    |   movel([0.283198, -1.182378, -2.685957, -0.844054, 1.570796, 1.853994],accel_mss,speed_ms,0,blend_radius_m)
    |   movel([0.283190, -1.181681, -2.686275, -0.844433, 1.570796, 1.853986],accel_mss,speed_ms,0,blend_radius_m)
    |   movel([0.283388, -1.180979, -2.686595, -0.844815, 1.570796, 1.854185],accel_mss,speed_ms,0,blend_radius_m)
    |   movel([0.283803, -1.180261, -2.686921, -0.845207, 1.570796, 1.854599],accel_mss,speed_ms,0,blend_radius_m)
    |   movel([0.284097, -1.179507, -2.687264, -0.845619, 1.570796, 1.854893],accel_mss,speed_ms,0,blend_radius_m)
    |   movel([0.284020, -1.179269, -2.687371, -0.845748, 1.570796, 1.854816],accel_mss,speed_ms,0,blend_radius_m)
    |   movel([0.283537, -1.179119, -2.687439, -0.845830, 1.570796, 1.854333],accel_mss,speed_ms,0,blend_radius_m)
    |   movel([0.283308, -1.178461, -2.687737, -0.846191, 1.570796, 1.854105],accel_mss,speed_ms,0,blend_radius_m)
    |   movel([0.283133, -1.176565, -2.688593, -0.847230, 1.570796, 1.853929],accel_mss,speed_ms,0,blend_radius_m)
    |   movel([0.283249, -1.175411, -2.689113, -0.847866, 1.570796, 1.854045],accel_mss,speed_ms,0,blend_radius_m)
    |   movel([0.283954, -1.172938, -2.690220, -0.849231, 1.570796, 1.854751],accel_mss,speed_ms,0,blend_radius_m)
    |   movel([0.284534, -1.171660, -2.690790, -0.849939, 1.570796, 1.855330],accel_mss,speed_ms,0,blend_radius_m)
    |   movel([0.286108, -1.169102, -2.691926, -0.851361, 1.570796, 1.856905],accel_mss,speed_ms,0,blend_radius_m)
    |   movel([0.287085, -1.167859, -2.692475, -0.852054, 1.570796, 1.857881],accel_mss,speed_ms,0,blend_radius_m)
    |   movel([0.288923, -1.165863, -2.693354, -0.853171, 1.570796, 1.859719],accel_mss,speed_ms,0,blend_radius_m)
    |   movel([0.289212, -1.165437, -2.693541, -0.853410, 1.570796, 1.860008],accel_mss,speed_ms,0,blend_radius_m)
    |   movel([0.289229, -1.165158, -2.693664, -0.853567, 1.570796, 1.860026],accel_mss,speed_ms,0,blend_radius_m)
    |   movel([0.288991, -1.164941, -2.693759, -0.853689, 1.570796, 1.859788],accel_mss,speed_ms,0,blend_radius_m)
    |   movel([0.288746, -1.164927, -2.693765, -0.853697, 1.570796, 1.859543],accel_mss,speed_ms,0,blend_radius_m)
    |   movel([0.288455, -1.165081, -2.693698, -0.853610, 1.570796, 1.859252],accel_mss,speed_ms,0,blend_radius_m)
    |   movel([0.287437, -1.165989, -2.693299, -0.853101, 1.570796, 1.858234],accel_mss,speed_ms,0,blend_radius_m)
    |   movel([0.286224, -1.167338, -2.692705, -0.852345, 1.570796, 1.857020],accel_mss,speed_ms,0,blend_radius_m)
    |   movel([0.285012, -1.168950, -2.691993, -0.851446, 1.570796, 1.855809],accel_mss,speed_ms,0,blend_radius_m)
    |   movel([0.283819, -1.170819, -2.691165, -0.850406, 1.570796, 1.854615],accel_mss,speed_ms,0,blend_radius_m)
    |   movel([0.282921, -1.172578, -2.690381, -0.849430, 1.570796, 1.853718],accel_mss,speed_ms,0,blend_radius_m)
    |   movel([0.282300, -1.174282, -2.689619, -0.848488, 1.570796, 1.853096],accel_mss,speed_ms,0,blend_radius_m)
    |   movel([0.281922, -1.175986, -2.688854, -0.847549, 1.570796, 1.852719],accel_mss,speed_ms,0,blend_radius_m)
    |   movel([0.281810, -1.177316, -2.688255, -0.846818, 1.570796, 1.852606],accel_mss,speed_ms,0,blend_radius_m)
    |   movel([0.281869, -1.178652, -2.687651, -0.846086, 1.570796, 1.852665],accel_mss,speed_ms,0,blend_radius_m)
    |   movel([0.282044, -1.179763, -2.687147, -0.845479, 1.570796, 1.852840],accel_mss,speed_ms,0,blend_radius_m)
    |   movel([0.282451, -1.180138, -2.686977, -0.845274, 1.570796, 1.853247],accel_mss,speed_ms,0,blend_radius_m)
    |   movel([0.282464, -1.180320, -2.686894, -0.845174, 1.570796, 1.853260],accel_mss,speed_ms,0,blend_radius_m)
    |   movel([0.281904, -1.182146, -2.686063, -0.844180, 1.570796, 1.852701],accel_mss,speed_ms,0,blend_radius_m)
    |   movel([0.281872, -1.183086, -2.685633, -0.843670, 1.570796, 1.852669],accel_mss,speed_ms,0,blend_radius_m)
    |   movel([0.282108, -1.183902, -2.685260, -0.843227, 1.570796, 1.852905],accel_mss,speed_ms,0,blend_radius_m)
    |   movel([0.282593, -1.184554, -2.684961, -0.842874, 1.570796, 1.853389],accel_mss,speed_ms,0,blend_radius_m)
    |   movel([0.283618, -1.185190, -2.684669, -0.842530, 1.570796, 1.854415],accel_mss,speed_ms,0,blend_radius_m)
    |   movel([0.284266, -1.185300, -2.684618, -0.842471, 1.570796, 1.855062],accel_mss,speed_ms,0,blend_radius_m)
    |   movel([0.285735, -1.185305, -2.684616, -0.842468, 1.570796, 1.856532],accel_mss,speed_ms,0,blend_radius_m)
    |   movel([0.286093, -1.185248, -2.684642, -0.842499, 1.570796, 1.856889],accel_mss,speed_ms,0,blend_radius_m)
    |   movel([0.286619, -1.184980, -2.684765, -0.842644, 1.570796, 1.857415],accel_mss,speed_ms,0,blend_radius_m)
    |   movel([0.286888, -1.184698, -2.684895, -0.842796, 1.570796, 1.857685],accel_mss,speed_ms,0,blend_radius_m)
    |   movel([0.287131, -1.184139, -2.685151, -0.843099, 1.570796, 1.857927],accel_mss,speed_ms,0,blend_radius_m)
    |   movel([0.287047, -1.183997, -2.685216, -0.843176, 1.570796, 1.857843],accel_mss,speed_ms,0,blend_radius_m)
    |   movel([0.285248, -1.183986, -2.685221, -0.843182, 1.570796, 1.856044],accel_mss,speed_ms,0,blend_radius_m)
    |   speed_ms = 0.005
    |   movel([0.285248, -1.174261, -2.680335, -0.857793, 1.570796, 1.856044],accel_mss,speed_ms,0,blend_radius_m)
    |   speed_ms = 0.040
    |   movel([0.315314, -1.140804, -2.694900, -0.876685, 1.570796, 1.886110],accel_mss,speed_ms,0,blend_radius_m)
    |   speed_ms = 0.005
    |   movel([0.315314, -1.150611, -2.699936, -0.861843, 1.570796, 1.886110],accel_mss,speed_ms,0,blend_radius_m)
    |   speed_ms = 0.025
    |   movel([0.314615, -1.150672, -2.699910, -0.861807, 1.570796, 1.885411],accel_mss,speed_ms,0,blend_radius_m)
    |   movel([0.314030, -1.150638, -2.699924, -0.861827, 1.570796, 1.884826],accel_mss,speed_ms,0,blend_radius_m)
    |   movel([0.311693, -1.150473, -2.699994, -0.861922, 1.570796, 1.882489],accel_mss,speed_ms,0,blend_radius_m)
    |   movel([0.309738, -1.150673, -2.699909, -0.861807, 1.570796, 1.880534],accel_mss,speed_ms,0,blend_radius_m)
    |   movel([0.307713, -1.151133, -2.699714, -0.861542, 1.570796, 1.878509],accel_mss,speed_ms,0,blend_radius_m)
    |   movel([0.305786, -1.151819, -2.699423, -0.861147, 1.570796, 1.876582],accel_mss,speed_ms,0,blend_radius_m)
    |   movel([0.303092, -1.153186, -2.698841, -0.860362, 1.570796, 1.873888],accel_mss,speed_ms,0,blend_radius_m)
    |   movel([0.300320, -1.155004, -2.698064, -0.859321, 1.570796, 1.871116],accel_mss,speed_ms,0,blend_radius_m)
    |   movel([0.297716, -1.157102, -2.697163, -0.858123, 1.570796, 1.868512],accel_mss,speed_ms,0,blend_radius_m)
    |   movel([0.295514, -1.159300, -2.696215, -0.856874, 1.570796, 1.866310],accel_mss,speed_ms,0,blend_radius_m)
    |   movel([0.294232, -1.160879, -2.695531, -0.855979, 1.570796, 1.865028],accel_mss,speed_ms,0,blend_radius_m)
    |   movel([0.293549, -1.162093, -2.695003, -0.855293, 1.570796, 1.864346],accel_mss,speed_ms,0,blend_radius_m)
    |   movel([0.293356, -1.163124, -2.694554, -0.854711, 1.570796, 1.864153],accel_mss,speed_ms,0,blend_radius_m)
    |   movel([0.293601, -1.164123, -2.694117, -0.854149, 1.570796, 1.864397],accel_mss,speed_ms,0,blend_radius_m)
    |   movel([0.293780, -1.164753, -2.693841, -0.853795, 1.570796, 1.864576],accel_mss,speed_ms,0,blend_radius_m)
    |   movel([0.293763, -1.165466, -2.693529, -0.853394, 1.570796, 1.864560],accel_mss,speed_ms,0,blend_radius_m)
    |   movel([0.293570, -1.166121, -2.693241, -0.853027, 1.570796, 1.864367],accel_mss,speed_ms,0,blend_radius_m)
    |   movel([0.293220, -1.166587, -2.693036, -0.852766, 1.570796, 1.864016],accel_mss,speed_ms,0,blend_radius_m)
    |   movel([0.292642, -1.167187, -2.692772, -0.852430, 1.570796, 1.863438],accel_mss,speed_ms,0,blend_radius_m)
    |   movel([0.292135, -1.167909, -2.692454, -0.852027, 1.570796, 1.862932],accel_mss,speed_ms,0,blend_radius_m)
    |   movel([0.291374, -1.169709, -2.691657, -0.851023, 1.570796, 1.862170],accel_mss,speed_ms,0,blend_radius_m)
    |   movel([0.291099, -1.170961, -2.691101, -0.850327, 1.570796, 1.861895],accel_mss,speed_ms,0,blend_radius_m)
    |   movel([0.291056, -1.172041, -2.690621, -0.849728, 1.570796, 1.861852],accel_mss,speed_ms,0,blend_radius_m)
    |   movel([0.291248, -1.172980, -2.690201, -0.849207, 1.570796, 1.862045],accel_mss,speed_ms,0,blend_radius_m)
    |   movel([0.292278, -1.174667, -2.689447, -0.848276, 1.570796, 1.863075],accel_mss,speed_ms,0,blend_radius_m)
    |   movel([0.291718, -1.176581, -2.688586, -0.847222, 1.570796, 1.862514],accel_mss,speed_ms,0,blend_radius_m)
    |   movel([0.291364, -1.178095, -2.687903, -0.846391, 1.570796, 1.862160],accel_mss,speed_ms,0,blend_radius_m)
    |   movel([0.291302, -1.179246, -2.687382, -0.845761, 1.570796, 1.862098],accel_mss,speed_ms,0,blend_radius_m)
    |   movel([0.291534, -1.180211, -2.686944, -0.845234, 1.570796, 1.862330],accel_mss,speed_ms,0,blend_radius_m)
    |   movel([0.292084, -1.181146, -2.686519, -0.844725, 1.570796, 1.862881],accel_mss,speed_ms,0,blend_radius_m)
    |   movel([0.292452, -1.181723, -2.686256, -0.844410, 1.570796, 1.863248],accel_mss,speed_ms,0,blend_radius_m)
    |   movel([0.292557, -1.182195, -2.686040, -0.844154, 1.570796, 1.863353],accel_mss,speed_ms,0,blend_radius_m)
    |   movel([0.292420, -1.182572, -2.685868, -0.843948, 1.570796, 1.863216],accel_mss,speed_ms,0,blend_radius_m)
    |   movel([0.292084, -1.182881, -2.685727, -0.843781, 1.570796, 1.862880],accel_mss,speed_ms,0,blend_radius_m)
    |   movel([0.291599, -1.182907, -2.685715, -0.843767, 1.570796, 1.862395],accel_mss,speed_ms,0,blend_radius_m)
    |   movel([0.290967, -1.182262, -2.686010, -0.844117, 1.570796, 1.861763],accel_mss,speed_ms,0,blend_radius_m)
    |   movel([0.290399, -1.181349, -2.686426, -0.844614, 1.570796, 1.861195],accel_mss,speed_ms,0,blend_radius_m)
    |   movel([0.290052, -1.180315, -2.686897, -0.845177, 1.570796, 1.860849],accel_mss,speed_ms,0,blend_radius_m)
    |   movel([0.289921, -1.178962, -2.687510, -0.845916, 1.570796, 1.860717],accel_mss,speed_ms,0,blend_radius_m)
    |   movel([0.290018, -1.178289, -2.687815, -0.846285, 1.570796, 1.860815],accel_mss,speed_ms,0,blend_radius_m)
    |   movel([0.290598, -1.175773, -2.688950, -0.847666, 1.570796, 1.861395],accel_mss,speed_ms,0,blend_radius_m)
    |   movel([0.290557, -1.175356, -2.689137, -0.847896, 1.570796, 1.861354],accel_mss,speed_ms,0,blend_radius_m)
    |   movel([0.289995, -1.174027, -2.689733, -0.848629, 1.570796, 1.860791],accel_mss,speed_ms,0,blend_radius_m)
    |   movel([0.289750, -1.173019, -2.690184, -0.849186, 1.570796, 1.860546],accel_mss,speed_ms,0,blend_radius_m)
    |   movel([0.289679, -1.171982, -2.690647, -0.849760, 1.570796, 1.860475],accel_mss,speed_ms,0,blend_radius_m)
    |   movel([0.289783, -1.170857, -2.691148, -0.850385, 1.570796, 1.860579],accel_mss,speed_ms,0,blend_radius_m)
    |   movel([0.290038, -1.169795, -2.691619, -0.850975, 1.570796, 1.860835],accel_mss,speed_ms,0,blend_radius_m)
    |   movel([0.290466, -1.168697, -2.692105, -0.851587, 1.570796, 1.861262],accel_mss,speed_ms,0,blend_radius_m)
    |   movel([0.291014, -1.167717, -2.692538, -0.852134, 1.570796, 1.861811],accel_mss,speed_ms,0,blend_radius_m)
    |   movel([0.291733, -1.166783, -2.692950, -0.852656, 1.570796, 1.862529],accel_mss,speed_ms,0,blend_radius_m)
    |   movel([0.292496, -1.165923, -2.693328, -0.853138, 1.570796, 1.863292],accel_mss,speed_ms,0,blend_radius_m)
    |   movel([0.292182, -1.164857, -2.693796, -0.853736, 1.570796, 1.862978],accel_mss,speed_ms,0,blend_radius_m)
    |   movel([0.292034, -1.163840, -2.694241, -0.854308, 1.570796, 1.862830],accel_mss,speed_ms,0,blend_radius_m)
    |   movel([0.292166, -1.162774, -2.694706, -0.854908, 1.570796, 1.862963],accel_mss,speed_ms,0,blend_radius_m)
    |   movel([0.292594, -1.161641, -2.695200, -0.855548, 1.570796, 1.863391],accel_mss,speed_ms,0,blend_radius_m)
    |   movel([0.293313, -1.160418, -2.695731, -0.856240, 1.570796, 1.864110],accel_mss,speed_ms,0,blend_radius_m)
    |   movel([0.294423, -1.159056, -2.696321, -0.857012, 1.570796, 1.865219],accel_mss,speed_ms,0,blend_radius_m)
    |   movel([0.296451, -1.157016, -2.697201, -0.858172, 1.570796, 1.867248],accel_mss,speed_ms,0,blend_radius_m)
    |   movel([0.298621, -1.155009, -2.698062, -0.859318, 1.570796, 1.869417],accel_mss,speed_ms,0,blend_radius_m)
    |   movel([0.300305, -1.153670, -2.698634, -0.860084, 1.570796, 1.871101],accel_mss,speed_ms,0,blend_radius_m)
    |   movel([0.302226, -1.152415, -2.699170, -0.860805, 1.570796, 1.873022],accel_mss,speed_ms,0,blend_radius_m)
    |   movel([0.304176, -1.151356, -2.699619, -0.861413, 1.570796, 1.874972],accel_mss,speed_ms,0,blend_radius_m)
    |   movel([0.306205, -1.150461, -2.699999, -0.861929, 1.570796, 1.877001],accel_mss,speed_ms,0,blend_radius_m)
    |   movel([0.308208, -1.149771, -2.700291, -0.862327, 1.570796, 1.879004],accel_mss,speed_ms,0,blend_radius_m)
    |   movel([0.310151, -1.149301, -2.700490, -0.862598, 1.570796, 1.880947],accel_mss,speed_ms,0,blend_radius_m)
    |   movel([0.312023, -1.149055, -2.700594, -0.862740, 1.570796, 1.882819],accel_mss,speed_ms,0,blend_radius_m)
    |   movel([0.313699, -1.149054, -2.700594, -0.862741, 1.570796, 1.884495],accel_mss,speed_ms,0,blend_radius_m)
    |   movel([0.315241, -1.149302, -2.700489, -0.862597, 1.570796, 1.886037],accel_mss,speed_ms,0,blend_radius_m)
    |   movel([0.315653, -1.149518, -2.700398, -0.862473, 1.570796, 1.886449],accel_mss,speed_ms,0,blend_radius_m)
    |   movel([0.315810, -1.149883, -2.700244, -0.862262, 1.570796, 1.886606],accel_mss,speed_ms,0,blend_radius_m)
    |   movel([0.315675, -1.150279, -2.700076, -0.862034, 1.570796, 1.886471],accel_mss,speed_ms,0,blend_radius_m)
    |   movel([0.315314, -1.150611, -2.699936, -0.861843, 1.570796, 1.886110],accel_mss,speed_ms,0,blend_radius_m)
    |   movel([0.314615, -1.150672, -2.699910, -0.861807, 1.570796, 1.885411],accel_mss,speed_ms,0,blend_radius_m)
    |   movel([0.314030, -1.150638, -2.699924, -0.861827, 1.570796, 1.884826],accel_mss,speed_ms,0,blend_radius_m)
    |   movel([0.312501, -1.150532, -2.699969, -0.861888, 1.570796, 1.883297],accel_mss,speed_ms,0,blend_radius_m)
    |   speed_ms = 0.005
    |   movel([0.312501, -1.140725, -2.694933, -0.876731, 1.570796, 1.883297],accel_mss,speed_ms,0,blend_radius_m)
    |   speed_ms = 0.040
    |   movel([0.330564, -1.150947, -2.690604, -0.870838, 1.570796, 1.901361],accel_mss,speed_ms,0,blend_radius_m)
    |   speed_ms = 0.005
    |   movel([0.330564, -1.160732, -2.695595, -0.856062, 1.570796, 1.901361],accel_mss,speed_ms,0,blend_radius_m)
    |   speed_ms = 0.025
    |   movel([0.330341, -1.160709, -2.695605, -0.856075, 1.570796, 1.901138],accel_mss,speed_ms,0,blend_radius_m)
    |   movel([0.329903, -1.160225, -2.695815, -0.856349, 1.570796, 1.900699],accel_mss,speed_ms,0,blend_radius_m)
    |   movel([0.327422, -1.156688, -2.697342, -0.858359, 1.570796, 1.898218],accel_mss,speed_ms,0,blend_radius_m)
    |   movel([0.325962, -1.154973, -2.698077, -0.859338, 1.570796, 1.896758],accel_mss,speed_ms,0,blend_radius_m)
    |   movel([0.324619, -1.153780, -2.698588, -0.860022, 1.570796, 1.895416],accel_mss,speed_ms,0,blend_radius_m)
    |   movel([0.323055, -1.152831, -2.698992, -0.860565, 1.570796, 1.893851],accel_mss,speed_ms,0,blend_radius_m)
    |   movel([0.321507, -1.152257, -2.699237, -0.860895, 1.570796, 1.892303],accel_mss,speed_ms,0,blend_radius_m)
    |   movel([0.319774, -1.151965, -2.699361, -0.861063, 1.570796, 1.890571],accel_mss,speed_ms,0,blend_radius_m)
    |   movel([0.317908, -1.151964, -2.699361, -0.861064, 1.570796, 1.888704],accel_mss,speed_ms,0,blend_radius_m)
    |   movel([0.315914, -1.152256, -2.699237, -0.860896, 1.570796, 1.886710],accel_mss,speed_ms,0,blend_radius_m)
    |   movel([0.313852, -1.152813, -2.699000, -0.860576, 1.570796, 1.884648],accel_mss,speed_ms,0,blend_radius_m)
    |   movel([0.312994, -1.153164, -2.698850, -0.860374, 1.570796, 1.883791],accel_mss,speed_ms,0,blend_radius_m)
    |   movel([0.309997, -1.154816, -2.698145, -0.859428, 1.570796, 1.880794],accel_mss,speed_ms,0,blend_radius_m)
    |   movel([0.308659, -1.155885, -2.697687, -0.858818, 1.570796, 1.879456],accel_mss,speed_ms,0,blend_radius_m)
    |   movel([0.307739, -1.157048, -2.697187, -0.858154, 1.570796, 1.878535],accel_mss,speed_ms,0,blend_radius_m)
    |   movel([0.307072, -1.158460, -2.696578, -0.857351, 1.570796, 1.877868],accel_mss,speed_ms,0,blend_radius_m)
    |   movel([0.306749, -1.159391, -2.696176, -0.856822, 1.570796, 1.877546],accel_mss,speed_ms,0,blend_radius_m)
    |   movel([0.305275, -1.159870, -2.695969, -0.856551, 1.570796, 1.876072],accel_mss,speed_ms,0,blend_radius_m)
    |   movel([0.303894, -1.160437, -2.695723, -0.856229, 1.570796, 1.874691],accel_mss,speed_ms,0,blend_radius_m)
    |   movel([0.302617, -1.161210, -2.695387, -0.855792, 1.570796, 1.873414],accel_mss,speed_ms,0,blend_radius_m)
    |   movel([0.301445, -1.162187, -2.694962, -0.855240, 1.570796, 1.872242],accel_mss,speed_ms,0,blend_radius_m)
    |   movel([0.300377, -1.163363, -2.694449, -0.854576, 1.570796, 1.871173],accel_mss,speed_ms,0,blend_radius_m)
    |   movel([0.299472, -1.164674, -2.693876, -0.853839, 1.570796, 1.870268],accel_mss,speed_ms,0,blend_radius_m)
    |   movel([0.299212, -1.165270, -2.693615, -0.853504, 1.570796, 1.870008],accel_mss,speed_ms,0,blend_radius_m)
    |   movel([0.298716, -1.167186, -2.692772, -0.852431, 1.570796, 1.869512],accel_mss,speed_ms,0,blend_radius_m)
    |   movel([0.298670, -1.168206, -2.692322, -0.851861, 1.570796, 1.869466],accel_mss,speed_ms,0,blend_radius_m)
    |   movel([0.298783, -1.169018, -2.691963, -0.851408, 1.570796, 1.869580],accel_mss,speed_ms,0,blend_radius_m)
    |   movel([0.299074, -1.169391, -2.691798, -0.851200, 1.570796, 1.869871],accel_mss,speed_ms,0,blend_radius_m)
    |   movel([0.299181, -1.169609, -2.691701, -0.851078, 1.570796, 1.869978],accel_mss,speed_ms,0,blend_radius_m)
    |   movel([0.299059, -1.169979, -2.691538, -0.850873, 1.570796, 1.869855],accel_mss,speed_ms,0,blend_radius_m)
    |   movel([0.298029, -1.171218, -2.690987, -0.850184, 1.570796, 1.868826],accel_mss,speed_ms,0,blend_radius_m)
    |   movel([0.297342, -1.171992, -2.690642, -0.849755, 1.570796, 1.868138],accel_mss,speed_ms,0,blend_radius_m)
    |   movel([0.296221, -1.173730, -2.689866, -0.848793, 1.570796, 1.867017],accel_mss,speed_ms,0,blend_radius_m)
    |   movel([0.295912, -1.174497, -2.689523, -0.848369, 1.570796, 1.866708],accel_mss,speed_ms,0,blend_radius_m)
    |   movel([0.295851, -1.176623, -2.688567, -0.847199, 1.570796, 1.866647],accel_mss,speed_ms,0,blend_radius_m)
    |   movel([0.295881, -1.177717, -2.688074, -0.846598, 1.570796, 1.866678],accel_mss,speed_ms,0,blend_radius_m)
    |   movel([0.295853, -1.180600, -2.686767, -0.845022, 1.570796, 1.866650],accel_mss,speed_ms,0,blend_radius_m)
    |   movel([0.295776, -1.180820, -2.686667, -0.844902, 1.570796, 1.866573],accel_mss,speed_ms,0,blend_radius_m)
    |   movel([0.295324, -1.181183, -2.686502, -0.844704, 1.570796, 1.866120],accel_mss,speed_ms,0,blend_radius_m)
    |   movel([0.295147, -1.181242, -2.686475, -0.844672, 1.570796, 1.865943],accel_mss,speed_ms,0,blend_radius_m)
    |   movel([0.294864, -1.181150, -2.686517, -0.844722, 1.570796, 1.865660],accel_mss,speed_ms,0,blend_radius_m)
    |   movel([0.294694, -1.180670, -2.686735, -0.844984, 1.570796, 1.865490],accel_mss,speed_ms,0,blend_radius_m)
    |   movel([0.294468, -1.177649, -2.688104, -0.846635, 1.570796, 1.865265],accel_mss,speed_ms,0,blend_radius_m)
    |   movel([0.294543, -1.175723, -2.688972, -0.847694, 1.570796, 1.865339],accel_mss,speed_ms,0,blend_radius_m)
    |   movel([0.294956, -1.173994, -2.689748, -0.848647, 1.570796, 1.865752],accel_mss,speed_ms,0,blend_radius_m)
    |   movel([0.295721, -1.172423, -2.690450, -0.849516, 1.570796, 1.866517],accel_mss,speed_ms,0,blend_radius_m)
    |   movel([0.296837, -1.170971, -2.691097, -0.850321, 1.570796, 1.867633],accel_mss,speed_ms,0,blend_radius_m)
    |   movel([0.297554, -1.170204, -2.691438, -0.850748, 1.570796, 1.868351],accel_mss,speed_ms,0,blend_radius_m)
    |   movel([0.297337, -1.167906, -2.692455, -0.852028, 1.570796, 1.868133],accel_mss,speed_ms,0,blend_radius_m)
    |   movel([0.297604, -1.166489, -2.693079, -0.852821, 1.570796, 1.868400],accel_mss,speed_ms,0,blend_radius_m)
    |   movel([0.298106, -1.165037, -2.693717, -0.853635, 1.570796, 1.868903],accel_mss,speed_ms,0,blend_radius_m)
    |   movel([0.298782, -1.163781, -2.694267, -0.854341, 1.570796, 1.869579],accel_mss,speed_ms,0,blend_radius_m)
    |   movel([0.300034, -1.162202, -2.694956, -0.855231, 1.570796, 1.870830],accel_mss,speed_ms,0,blend_radius_m)
    |   movel([0.301657, -1.160695, -2.695611, -0.856083, 1.570796, 1.872454],accel_mss,speed_ms,0,blend_radius_m)
    |   movel([0.303428, -1.159450, -2.696151, -0.856789, 1.570796, 1.874224],accel_mss,speed_ms,0,blend_radius_m)
    |   movel([0.305117, -1.158647, -2.696498, -0.857245, 1.570796, 1.875913],accel_mss,speed_ms,0,blend_radius_m)
    |   movel([0.305966, -1.158277, -2.696657, -0.857454, 1.570796, 1.876763],accel_mss,speed_ms,0,blend_radius_m)
    |   movel([0.306111, -1.158107, -2.696731, -0.857551, 1.570796, 1.876908],accel_mss,speed_ms,0,blend_radius_m)
    |   movel([0.306523, -1.156986, -2.697214, -0.858190, 1.570796, 1.877319],accel_mss,speed_ms,0,blend_radius_m)
    |   movel([0.306747, -1.156613, -2.697374, -0.858402, 1.570796, 1.877544],accel_mss,speed_ms,0,blend_radius_m)
    |   movel([0.307476, -1.155654, -2.697785, -0.858949, 1.570796, 1.878273],accel_mss,speed_ms,0,blend_radius_m)
    |   movel([0.308347, -1.154796, -2.698153, -0.859440, 1.570796, 1.879144],accel_mss,speed_ms,0,blend_radius_m)
    |   movel([0.309487, -1.153902, -2.698535, -0.859951, 1.570796, 1.880283],accel_mss,speed_ms,0,blend_radius_m)
    |   movel([0.310666, -1.153129, -2.698865, -0.860395, 1.570796, 1.881462],accel_mss,speed_ms,0,blend_radius_m)
    |   movel([0.312068, -1.152374, -2.699187, -0.860828, 1.570796, 1.882864],accel_mss,speed_ms,0,blend_radius_m)
    |   movel([0.313470, -1.151766, -2.699446, -0.861178, 1.570796, 1.884266],accel_mss,speed_ms,0,blend_radius_m)
    |   movel([0.316489, -1.150865, -2.699828, -0.861696, 1.570796, 1.887286],accel_mss,speed_ms,0,blend_radius_m)
    |   movel([0.318328, -1.150563, -2.699956, -0.861870, 1.570796, 1.889125],accel_mss,speed_ms,0,blend_radius_m)
    |   movel([0.319922, -1.150503, -2.699981, -0.861905, 1.570796, 1.890719],accel_mss,speed_ms,0,blend_radius_m)
    |   movel([0.321440, -1.150681, -2.699906, -0.861802, 1.570796, 1.892236],accel_mss,speed_ms,0,blend_radius_m)
    |   movel([0.323038, -1.151114, -2.699722, -0.861553, 1.570796, 1.893835],accel_mss,speed_ms,0,blend_radius_m)
    |   movel([0.324964, -1.151992, -2.699349, -0.861048, 1.570796, 1.895760],accel_mss,speed_ms,0,blend_radius_m)
    |   movel([0.326646, -1.153232, -2.698822, -0.860336, 1.570796, 1.897442],accel_mss,speed_ms,0,blend_radius_m)
    |   movel([0.328267, -1.155000, -2.698066, -0.859323, 1.570796, 1.899063],accel_mss,speed_ms,0,blend_radius_m)
    |   movel([0.330866, -1.158912, -2.696383, -0.857094, 1.570796, 1.901662],accel_mss,speed_ms,0,blend_radius_m)
    |   movel([0.331156, -1.159778, -2.696008, -0.856603, 1.570796, 1.901953],accel_mss,speed_ms,0,blend_radius_m)
    |   movel([0.331017, -1.160335, -2.695767, -0.856287, 1.570796, 1.901813],accel_mss,speed_ms,0,blend_radius_m)
    |   movel([0.330564, -1.160732, -2.695595, -0.856062, 1.570796, 1.901361],accel_mss,speed_ms,0,blend_radius_m)
    |   movel([0.330341, -1.160709, -2.695605, -0.856075, 1.570796, 1.901138],accel_mss,speed_ms,0,blend_radius_m)
    |   movel([0.329903, -1.160225, -2.695815, -0.856349, 1.570796, 1.900699],accel_mss,speed_ms,0,blend_radius_m)
    |   movel([0.329043, -1.158994, -2.696348, -0.857047, 1.570796, 1.899840],accel_mss,speed_ms,0,blend_radius_m)
    |   speed_ms = 0.005
    |   movel([0.329043, -1.149205, -2.691349, -0.871835, 1.570796, 1.899840],accel_mss,speed_ms,0,blend_radius_m)
    |   speed_ms = 0.040
    |   movel([0.331713, -1.158475, -2.687349, -0.866565, 1.570796, 1.902510],accel_mss,speed_ms,0,blend_radius_m)
    |   speed_ms = 0.005
    |   movel([0.331713, -1.168242, -2.692306, -0.851841, 1.570796, 1.902510],accel_mss,speed_ms,0,blend_radius_m)
    |   speed_ms = 0.025
    |   movel([0.331306, -1.168113, -2.692363, -0.851912, 1.570796, 1.902103],accel_mss,speed_ms,0,blend_radius_m)
    |   movel([0.331181, -1.167790, -2.692506, -0.852093, 1.570796, 1.901977],accel_mss,speed_ms,0,blend_radius_m)
    |   movel([0.330488, -1.165082, -2.693697, -0.853610, 1.570796, 1.901285],accel_mss,speed_ms,0,blend_radius_m)
    |   movel([0.329418, -1.163092, -2.694568, -0.854729, 1.570796, 1.900215],accel_mss,speed_ms,0,blend_radius_m)
    |   movel([0.327976, -1.161415, -2.695298, -0.855676, 1.570796, 1.898772],accel_mss,speed_ms,0,blend_radius_m)
    |   movel([0.326286, -1.160232, -2.695812, -0.856345, 1.570796, 1.897083],accel_mss,speed_ms,0,blend_radius_m)
    |   movel([0.325017, -1.159721, -2.696033, -0.856635, 1.570796, 1.895813],accel_mss,speed_ms,0,blend_radius_m)
    |   movel([0.323332, -1.159309, -2.696211, -0.856869, 1.570796, 1.894129],accel_mss,speed_ms,0,blend_radius_m)
    |   movel([0.321666, -1.159053, -2.696322, -0.857014, 1.570796, 1.892462],accel_mss,speed_ms,0,blend_radius_m)
    |   movel([0.320604, -1.159119, -2.696294, -0.856976, 1.570796, 1.891400],accel_mss,speed_ms,0,blend_radius_m)
    |   movel([0.319128, -1.159715, -2.696036, -0.856638, 1.570796, 1.889924],accel_mss,speed_ms,0,blend_radius_m)
    |   movel([0.318351, -1.160251, -2.695804, -0.856335, 1.570796, 1.889148],accel_mss,speed_ms,0,blend_radius_m)
    |   movel([0.316474, -1.161927, -2.695075, -0.855386, 1.570796, 1.887270],accel_mss,speed_ms,0,blend_radius_m)
    |   movel([0.313923, -1.162515, -2.694819, -0.855054, 1.570796, 1.884719],accel_mss,speed_ms,0,blend_radius_m)
    |   movel([0.311493, -1.163182, -2.694529, -0.854679, 1.570796, 1.882289],accel_mss,speed_ms,0,blend_radius_m)
    |   movel([0.310725, -1.163546, -2.694369, -0.854473, 1.570796, 1.881521],accel_mss,speed_ms,0,blend_radius_m)
    |   movel([0.308314, -1.165097, -2.693690, -0.853601, 1.570796, 1.879110],accel_mss,speed_ms,0,blend_radius_m)
    |   movel([0.307457, -1.165878, -2.693348, -0.853163, 1.570796, 1.878254],accel_mss,speed_ms,0,blend_radius_m)
    |   movel([0.306883, -1.166716, -2.692979, -0.852694, 1.570796, 1.877680],accel_mss,speed_ms,0,blend_radius_m)
    |   movel([0.306453, -1.167771, -2.692514, -0.852104, 1.570796, 1.877249],accel_mss,speed_ms,0,blend_radius_m)
    |   movel([0.306245, -1.168703, -2.692103, -0.851583, 1.570796, 1.877041],accel_mss,speed_ms,0,blend_radius_m)
    |   movel([0.306317, -1.168871, -2.692028, -0.851490, 1.570796, 1.877113],accel_mss,speed_ms,0,blend_radius_m)
    |   movel([0.306750, -1.169089, -2.691932, -0.851368, 1.570796, 1.877546],accel_mss,speed_ms,0,blend_radius_m)
    |   movel([0.306794, -1.169237, -2.691866, -0.851286, 1.570796, 1.877590],accel_mss,speed_ms,0,blend_radius_m)
    |   movel([0.306593, -1.169712, -2.691656, -0.851021, 1.570796, 1.877390],accel_mss,speed_ms,0,blend_radius_m)
    |   movel([0.306273, -1.169988, -2.691533, -0.850867, 1.570796, 1.877070],accel_mss,speed_ms,0,blend_radius_m)
    |   movel([0.304136, -1.171018, -2.691076, -0.850295, 1.570796, 1.874933],accel_mss,speed_ms,0,blend_radius_m)
    |   movel([0.303280, -1.171628, -2.690804, -0.849956, 1.570796, 1.874076],accel_mss,speed_ms,0,blend_radius_m)
    |   movel([0.301531, -1.173235, -2.690087, -0.849066, 1.570796, 1.872327],accel_mss,speed_ms,0,blend_radius_m)
    |   movel([0.301020, -1.173828, -2.689822, -0.848738, 1.570796, 1.871816],accel_mss,speed_ms,0,blend_radius_m)
    |   movel([0.300389, -1.174911, -2.689337, -0.848141, 1.570796, 1.871186],accel_mss,speed_ms,0,blend_radius_m)
    |   movel([0.300062, -1.175767, -2.688952, -0.847669, 1.570796, 1.870858],accel_mss,speed_ms,0,blend_radius_m)
    |   movel([0.299607, -1.177615, -2.688120, -0.846654, 1.570796, 1.870404],accel_mss,speed_ms,0,blend_radius_m)
    |   movel([0.299612, -1.178043, -2.687926, -0.846420, 1.570796, 1.870409],accel_mss,speed_ms,0,blend_radius_m)
    |   movel([0.299615, -1.178734, -2.687614, -0.846041, 1.570796, 1.870411],accel_mss,speed_ms,0,blend_radius_m)
    |   movel([0.299503, -1.178945, -2.687518, -0.845926, 1.570796, 1.870299],accel_mss,speed_ms,0,blend_radius_m)
    |   movel([0.298972, -1.179400, -2.687312, -0.845677, 1.570796, 1.869769],accel_mss,speed_ms,0,blend_radius_m)
    |   movel([0.298670, -1.179460, -2.687285, -0.845644, 1.570796, 1.869466],accel_mss,speed_ms,0,blend_radius_m)
    |   movel([0.298302, -1.179128, -2.687435, -0.845825, 1.570796, 1.869098],accel_mss,speed_ms,0,blend_radius_m)
    |   movel([0.298322, -1.178019, -2.687937, -0.846433, 1.570796, 1.869118],accel_mss,speed_ms,0,blend_radius_m)
    |   movel([0.299097, -1.175195, -2.689210, -0.847985, 1.570796, 1.869893],accel_mss,speed_ms,0,blend_radius_m)
    |   movel([0.299377, -1.174512, -2.689516, -0.848361, 1.570796, 1.870173],accel_mss,speed_ms,0,blend_radius_m)
    |   movel([0.300237, -1.173205, -2.690101, -0.849083, 1.570796, 1.871033],accel_mss,speed_ms,0,blend_radius_m)
    |   movel([0.301128, -1.172172, -2.690562, -0.849655, 1.570796, 1.871924],accel_mss,speed_ms,0,blend_radius_m)
    |   movel([0.302132, -1.171214, -2.690989, -0.850186, 1.570796, 1.872929],accel_mss,speed_ms,0,blend_radius_m)
    |   movel([0.303176, -1.170393, -2.691354, -0.850642, 1.570796, 1.873972],accel_mss,speed_ms,0,blend_radius_m)
    |   movel([0.304919, -1.169330, -2.691825, -0.851234, 1.570796, 1.875715],accel_mss,speed_ms,0,blend_radius_m)
    |   movel([0.305106, -1.169138, -2.691910, -0.851341, 1.570796, 1.875903],accel_mss,speed_ms,0,blend_radius_m)
    |   movel([0.305251, -1.168250, -2.692303, -0.851836, 1.570796, 1.876047],accel_mss,speed_ms,0,blend_radius_m)
    |   movel([0.305493, -1.167355, -2.692698, -0.852336, 1.570796, 1.876289],accel_mss,speed_ms,0,blend_radius_m)
    |   movel([0.305832, -1.166483, -2.693082, -0.852824, 1.570796, 1.876628],accel_mss,speed_ms,0,blend_radius_m)
    |   movel([0.306211, -1.165835, -2.693367, -0.853187, 1.570796, 1.877008],accel_mss,speed_ms,0,blend_radius_m)
    |   movel([0.306836, -1.165086, -2.693695, -0.853608, 1.570796, 1.877632],accel_mss,speed_ms,0,blend_radius_m)
    |   movel([0.307551, -1.164418, -2.693988, -0.853983, 1.570796, 1.878347],accel_mss,speed_ms,0,blend_radius_m)
    |   movel([0.309421, -1.163106, -2.694562, -0.854721, 1.570796, 1.880217],accel_mss,speed_ms,0,blend_radius_m)
    |   movel([0.311698, -1.161982, -2.695052, -0.855356, 1.570796, 1.882494],accel_mss,speed_ms,0,blend_radius_m)
    |   movel([0.316256, -1.160519, -2.695688, -0.856183, 1.570796, 1.887052],accel_mss,speed_ms,0,blend_radius_m)
    |   movel([0.316728, -1.160293, -2.695785, -0.856311, 1.570796, 1.887525],accel_mss,speed_ms,0,blend_radius_m)
    |   movel([0.317927, -1.159215, -2.696252, -0.856922, 1.570796, 1.888723],accel_mss,speed_ms,0,blend_radius_m)
    |   movel([0.318329, -1.158914, -2.696382, -0.857093, 1.570796, 1.889125],accel_mss,speed_ms,0,blend_radius_m)
    |   movel([0.319436, -1.158287, -2.696653, -0.857449, 1.570796, 1.890232],accel_mss,speed_ms,0,blend_radius_m)
    |   movel([0.320040, -1.158088, -2.696739, -0.857562, 1.570796, 1.890837],accel_mss,speed_ms,0,blend_radius_m)
    |   movel([0.320882, -1.157898, -2.696821, -0.857670, 1.570796, 1.891679],accel_mss,speed_ms,0,blend_radius_m)
    |   movel([0.322944, -1.157677, -2.696916, -0.857796, 1.570796, 1.893740],accel_mss,speed_ms,0,blend_radius_m)
    |   movel([0.324806, -1.157871, -2.696832, -0.857686, 1.570796, 1.895602],accel_mss,speed_ms,0,blend_radius_m)
    |   movel([0.326669, -1.158486, -2.696567, -0.857336, 1.570796, 1.897466],accel_mss,speed_ms,0,blend_radius_m)
    |   movel([0.328292, -1.159413, -2.696166, -0.856809, 1.570796, 1.899088],accel_mss,speed_ms,0,blend_radius_m)
    |   movel([0.329758, -1.160703, -2.695607, -0.856078, 1.570796, 1.900554],accel_mss,speed_ms,0,blend_radius_m)
    |   movel([0.330942, -1.162270, -2.694926, -0.855193, 1.570796, 1.901738],accel_mss,speed_ms,0,blend_radius_m)
    |   movel([0.331828, -1.164089, -2.694132, -0.854168, 1.570796, 1.902624],accel_mss,speed_ms,0,blend_radius_m)
    |   movel([0.332407, -1.166129, -2.693237, -0.853022, 1.570796, 1.903203],accel_mss,speed_ms,0,blend_radius_m)
    |   movel([0.332496, -1.166919, -2.692890, -0.852580, 1.570796, 1.903292],accel_mss,speed_ms,0,blend_radius_m)
    |   movel([0.332398, -1.167537, -2.692618, -0.852234, 1.570796, 1.903194],accel_mss,speed_ms,0,blend_radius_m)
    |   movel([0.332125, -1.167972, -2.692426, -0.851991, 1.570796, 1.902922],accel_mss,speed_ms,0,blend_radius_m)
    |   movel([0.331713, -1.168242, -2.692306, -0.851841, 1.570796, 1.902510],accel_mss,speed_ms,0,blend_radius_m)
    |   movel([0.331306, -1.168113, -2.692363, -0.851912, 1.570796, 1.902103],accel_mss,speed_ms,0,blend_radius_m)
    |   movel([0.331181, -1.167790, -2.692506, -0.852093, 1.570796, 1.901977],accel_mss,speed_ms,0,blend_radius_m)
    |   movel([0.330747, -1.166094, -2.693253, -0.853042, 1.570796, 1.901543],accel_mss,speed_ms,0,blend_radius_m)
    |   speed_ms = 0.005
    |   movel([0.330747, -1.156321, -2.688286, -0.867781, 1.570796, 1.901543],accel_mss,speed_ms,0,blend_radius_m)
    |   speed_ms = 0.040
    |   movel([0.331469, -1.169115, -2.682650, -0.860624, 1.570796, 1.902266],accel_mss,speed_ms,0,blend_radius_m)
    |   speed_ms = 0.005
    |   movel([0.331469, -1.178854, -2.687559, -0.845975, 1.570796, 1.902266],accel_mss,speed_ms,0,blend_radius_m)
    |   speed_ms = 0.025
    |   movel([0.330682, -1.179241, -2.687384, -0.845764, 1.570796, 1.901478],accel_mss,speed_ms,0,blend_radius_m)
    |   movel([0.330527, -1.179246, -2.687382, -0.845761, 1.570796, 1.901324],accel_mss,speed_ms,0,blend_radius_m)
    |   movel([0.330285, -1.179088, -2.687453, -0.845847, 1.570796, 1.901081],accel_mss,speed_ms,0,blend_radius_m)
    |   movel([0.330236, -1.178791, -2.687588, -0.846010, 1.570796, 1.901032],accel_mss,speed_ms,0,blend_radius_m)
    |   movel([0.330383, -1.178440, -2.687747, -0.846202, 1.570796, 1.901179],accel_mss,speed_ms,0,blend_radius_m)
    |   movel([0.330690, -1.178117, -2.687893, -0.846379, 1.570796, 1.901487],accel_mss,speed_ms,0,blend_radius_m)
    |   movel([0.331117, -1.177631, -2.688113, -0.846646, 1.570796, 1.901914],accel_mss,speed_ms,0,blend_radius_m)
    |   movel([0.331243, -1.177291, -2.688266, -0.846832, 1.570796, 1.902040],accel_mss,speed_ms,0,blend_radius_m)
    |   movel([0.331366, -1.176749, -2.688511, -0.847130, 1.570796, 1.902162],accel_mss,speed_ms,0,blend_radius_m)
    |   movel([0.331570, -1.174446, -2.689546, -0.848397, 1.570796, 1.902366],accel_mss,speed_ms,0,blend_radius_m)
    |   movel([0.331243, -1.172459, -2.690434, -0.849496, 1.570796, 1.902040],accel_mss,speed_ms,0,blend_radius_m)
    |   movel([0.330392, -1.170834, -2.691158, -0.850397, 1.570796, 1.901188],accel_mss,speed_ms,0,blend_radius_m)
    |   movel([0.329032, -1.169616, -2.691698, -0.851074, 1.570796, 1.899828],accel_mss,speed_ms,0,blend_radius_m)
    |   movel([0.328083, -1.169161, -2.691900, -0.851328, 1.570796, 1.898879],accel_mss,speed_ms,0,blend_radius_m)
    |   movel([0.325708, -1.168715, -2.692097, -0.851577, 1.570796, 1.896504],accel_mss,speed_ms,0,blend_radius_m)
    |   movel([0.324679, -1.168798, -2.692061, -0.851531, 1.570796, 1.895475],accel_mss,speed_ms,0,blend_radius_m)
    |   movel([0.323933, -1.169040, -2.691953, -0.851395, 1.570796, 1.894730],accel_mss,speed_ms,0,blend_radius_m)
    |   movel([0.323752, -1.169240, -2.691865, -0.851284, 1.570796, 1.894548],accel_mss,speed_ms,0,blend_radius_m)
    |   movel([0.323250, -1.170060, -2.691501, -0.850827, 1.570796, 1.894046],accel_mss,speed_ms,0,blend_radius_m)
    |   movel([0.322821, -1.170309, -2.691391, -0.850689, 1.570796, 1.893618],accel_mss,speed_ms,0,blend_radius_m)
    |   movel([0.322188, -1.170348, -2.691374, -0.850667, 1.570796, 1.892984],accel_mss,speed_ms,0,blend_radius_m)
    |   movel([0.321130, -1.170170, -2.691453, -0.850767, 1.570796, 1.891926],accel_mss,speed_ms,0,blend_radius_m)
    |   movel([0.319263, -1.170120, -2.691475, -0.850794, 1.570796, 1.890059],accel_mss,speed_ms,0,blend_radius_m)
    |   movel([0.318553, -1.170236, -2.691423, -0.850729, 1.570796, 1.889350],accel_mss,speed_ms,0,blend_radius_m)
    |   movel([0.316685, -1.170740, -2.691199, -0.850449, 1.570796, 1.887481],accel_mss,speed_ms,0,blend_radius_m)
    |   movel([0.315326, -1.171430, -2.690893, -0.850066, 1.570796, 1.886122],accel_mss,speed_ms,0,blend_radius_m)
    |   movel([0.314393, -1.172331, -2.690491, -0.849566, 1.570796, 1.885189],accel_mss,speed_ms,0,blend_radius_m)
    |   movel([0.313800, -1.173463, -2.689986, -0.848940, 1.570796, 1.884596],accel_mss,speed_ms,0,blend_radius_m)
    |   movel([0.313494, -1.174437, -2.689549, -0.848402, 1.570796, 1.884291],accel_mss,speed_ms,0,blend_radius_m)
    |   movel([0.312668, -1.174607, -2.689473, -0.848309, 1.570796, 1.883464],accel_mss,speed_ms,0,blend_radius_m)
    |   movel([0.311909, -1.174837, -2.689370, -0.848182, 1.570796, 1.882705],accel_mss,speed_ms,0,blend_radius_m)
    |   movel([0.311134, -1.175217, -2.689200, -0.847972, 1.570796, 1.881930],accel_mss,speed_ms,0,blend_radius_m)
    |   movel([0.309598, -1.176378, -2.688677, -0.847333, 1.570796, 1.880394],accel_mss,speed_ms,0,blend_radius_m)
    |   movel([0.308951, -1.177067, -2.688367, -0.846955, 1.570796, 1.879747],accel_mss,speed_ms,0,blend_radius_m)
    |   movel([0.308397, -1.177815, -2.688030, -0.846545, 1.570796, 1.879194],accel_mss,speed_ms,0,blend_radius_m)
    |   movel([0.308016, -1.178523, -2.687709, -0.846157, 1.570796, 1.878812],accel_mss,speed_ms,0,blend_radius_m)
    |   movel([0.307480, -1.180072, -2.687007, -0.845310, 1.570796, 1.878276],accel_mss,speed_ms,0,blend_radius_m)
    |   movel([0.307253, -1.180364, -2.686874, -0.845151, 1.570796, 1.878050],accel_mss,speed_ms,0,blend_radius_m)
    |   movel([0.306952, -1.180575, -2.686778, -0.845036, 1.570796, 1.877749],accel_mss,speed_ms,0,blend_radius_m)
    |   movel([0.306688, -1.180630, -2.686754, -0.845006, 1.570796, 1.877485],accel_mss,speed_ms,0,blend_radius_m)
    |   movel([0.306514, -1.180523, -2.686802, -0.845064, 1.570796, 1.877310],accel_mss,speed_ms,0,blend_radius_m)
    |   movel([0.306409, -1.179886, -2.687092, -0.845412, 1.570796, 1.877206],accel_mss,speed_ms,0,blend_radius_m)
    |   movel([0.306585, -1.179075, -2.687459, -0.845855, 1.570796, 1.877381],accel_mss,speed_ms,0,blend_radius_m)
    |   movel([0.306955, -1.178226, -2.687844, -0.846319, 1.570796, 1.877751],accel_mss,speed_ms,0,blend_radius_m)
    |   movel([0.307530, -1.177295, -2.688264, -0.846830, 1.570796, 1.878326],accel_mss,speed_ms,0,blend_radius_m)
    |   movel([0.308227, -1.176405, -2.688665, -0.847318, 1.570796, 1.879023],accel_mss,speed_ms,0,blend_radius_m)
    |   movel([0.309047, -1.175553, -2.689049, -0.847787, 1.570796, 1.879843],accel_mss,speed_ms,0,blend_radius_m)
    |   movel([0.309945, -1.174793, -2.689390, -0.848206, 1.570796, 1.880741],accel_mss,speed_ms,0,blend_radius_m)
    |   movel([0.310844, -1.174197, -2.689657, -0.848535, 1.570796, 1.881640],accel_mss,speed_ms,0,blend_radius_m)
    |   movel([0.311760, -1.173751, -2.689857, -0.848781, 1.570796, 1.882556],accel_mss,speed_ms,0,blend_radius_m)
    |   movel([0.312381, -1.173381, -2.690023, -0.848986, 1.570796, 1.883177],accel_mss,speed_ms,0,blend_radius_m)
    |   movel([0.312612, -1.173117, -2.690140, -0.849131, 1.570796, 1.883408],accel_mss,speed_ms,0,blend_radius_m)
    |   movel([0.313295, -1.172066, -2.690609, -0.849713, 1.570796, 1.884092],accel_mss,speed_ms,0,blend_radius_m)
    |   movel([0.313953, -1.171357, -2.690925, -0.850107, 1.570796, 1.884749],accel_mss,speed_ms,0,blend_radius_m)
    |   movel([0.315643, -1.170069, -2.691497, -0.850822, 1.570796, 1.886439],accel_mss,speed_ms,0,blend_radius_m)
    |   movel([0.316858, -1.169488, -2.691755, -0.851146, 1.570796, 1.887654],accel_mss,speed_ms,0,blend_radius_m)
    |   movel([0.318433, -1.169018, -2.691963, -0.851408, 1.570796, 1.889230],accel_mss,speed_ms,0,blend_radius_m)
    |   movel([0.320036, -1.168735, -2.692088, -0.851566, 1.570796, 1.890833],accel_mss,speed_ms,0,blend_radius_m)
    |   movel([0.322567, -1.168740, -2.692086, -0.851563, 1.570796, 1.893364],accel_mss,speed_ms,0,blend_radius_m)
    |   movel([0.322872, -1.168592, -2.692151, -0.851645, 1.570796, 1.893669],accel_mss,speed_ms,0,blend_radius_m)
    |   movel([0.324135, -1.167670, -2.692559, -0.852160, 1.570796, 1.894931],accel_mss,speed_ms,0,blend_radius_m)
    |   movel([0.324975, -1.167402, -2.692677, -0.852310, 1.570796, 1.895771],accel_mss,speed_ms,0,blend_radius_m)
    |   movel([0.327374, -1.167417, -2.692670, -0.852301, 1.570796, 1.898171],accel_mss,speed_ms,0,blend_radius_m)
    |   movel([0.328614, -1.167684, -2.692553, -0.852152, 1.570796, 1.899410],accel_mss,speed_ms,0,blend_radius_m)
    |   movel([0.329739, -1.168112, -2.692364, -0.851913, 1.570796, 1.900535],accel_mss,speed_ms,0,blend_radius_m)
    |   movel([0.330655, -1.168678, -2.692114, -0.851597, 1.570796, 1.901451],accel_mss,speed_ms,0,blend_radius_m)
    |   movel([0.331414, -1.169411, -2.691789, -0.851189, 1.570796, 1.902210],accel_mss,speed_ms,0,blend_radius_m)
    |   movel([0.332359, -1.171022, -2.691074, -0.850293, 1.570796, 1.903155],accel_mss,speed_ms,0,blend_radius_m)
    |   movel([0.332853, -1.172983, -2.690200, -0.849206, 1.570796, 1.903649],accel_mss,speed_ms,0,blend_radius_m)
    |   movel([0.332875, -1.175166, -2.689222, -0.848000, 1.570796, 1.903671],accel_mss,speed_ms,0,blend_radius_m)
    |   movel([0.332415, -1.177444, -2.688197, -0.846748, 1.570796, 1.903211],accel_mss,speed_ms,0,blend_radius_m)
    |   movel([0.332236, -1.177958, -2.687965, -0.846466, 1.570796, 1.903033],accel_mss,speed_ms,0,blend_radius_m)
    |   movel([0.331821, -1.178571, -2.687687, -0.846130, 1.570796, 1.902617],accel_mss,speed_ms,0,blend_radius_m)
    |   movel([0.331469, -1.178854, -2.687559, -0.845975, 1.570796, 1.902266],accel_mss,speed_ms,0,blend_radius_m)
    |   movel([0.330682, -1.179241, -2.687384, -0.845764, 1.570796, 1.901478],accel_mss,speed_ms,0,blend_radius_m)
    |   movel([0.330527, -1.179246, -2.687382, -0.845761, 1.570796, 1.901324],accel_mss,speed_ms,0,blend_radius_m)
    |   movel([0.330285, -1.179088, -2.687453, -0.845847, 1.570796, 1.901081],accel_mss,speed_ms,0,blend_radius_m)
    |   movel([0.330236, -1.178791, -2.687588, -0.846010, 1.570796, 1.901032],accel_mss,speed_ms,0,blend_radius_m)
    |   movel([0.330383, -1.178440, -2.687747, -0.846202, 1.570796, 1.901179],accel_mss,speed_ms,0,blend_radius_m)
    |   movel([0.330690, -1.178117, -2.687893, -0.846379, 1.570796, 1.901487],accel_mss,speed_ms,0,blend_radius_m)
    |   movel([0.331117, -1.177631, -2.688113, -0.846646, 1.570796, 1.901914],accel_mss,speed_ms,0,blend_radius_m)
    |   movel([0.331194, -1.177425, -2.688206, -0.846759, 1.570796, 1.901990],accel_mss,speed_ms,0,blend_radius_m)
    |   speed_ms = 0.005
    |   movel([0.331194, -1.167681, -2.683290, -0.861418, 1.570796, 1.901990],accel_mss,speed_ms,0,blend_radius_m)
    |   speed_ms = 0.040
    |   movel([0.330295, -1.185364, -2.675246, -0.851779, 1.570796, 1.901092],accel_mss,speed_ms,0,blend_radius_m)
    |   speed_ms = 0.005
    |   movel([0.330295, -1.195055, -2.680082, -0.837252, 1.570796, 1.901092],accel_mss,speed_ms,0,blend_radius_m)
    |   speed_ms = 0.025
    |   movel([0.330668, -1.194304, -2.680435, -0.837650, 1.570796, 1.901464],accel_mss,speed_ms,0,blend_radius_m)
    |   movel([0.331756, -1.190620, -2.682157, -0.839612, 1.570796, 1.902552],accel_mss,speed_ms,0,blend_radius_m)
    |   movel([0.332001, -1.189344, -2.682750, -0.840295, 1.570796, 1.902797],accel_mss,speed_ms,0,blend_radius_m)
    |   movel([0.332119, -1.187217, -2.683735, -0.841437, 1.570796, 1.902916],accel_mss,speed_ms,0,blend_radius_m)
    |   movel([0.331930, -1.185198, -2.684665, -0.842526, 1.570796, 1.902726],accel_mss,speed_ms,0,blend_radius_m)
    |   movel([0.331458, -1.183462, -2.685461, -0.843466, 1.570796, 1.902255],accel_mss,speed_ms,0,blend_radius_m)
    |   movel([0.330731, -1.182191, -2.686042, -0.844156, 1.570796, 1.901527],accel_mss,speed_ms,0,blend_radius_m)
    |   movel([0.329629, -1.181311, -2.686443, -0.844634, 1.570796, 1.900425],accel_mss,speed_ms,0,blend_radius_m)
    |   movel([0.328223, -1.180944, -2.686610, -0.844834, 1.570796, 1.899019],accel_mss,speed_ms,0,blend_radius_m)
    |   movel([0.326708, -1.181131, -2.686525, -0.844733, 1.570796, 1.897505],accel_mss,speed_ms,0,blend_radius_m)
    |   movel([0.325994, -1.181415, -2.686396, -0.844578, 1.570796, 1.896790],accel_mss,speed_ms,0,blend_radius_m)
    |   movel([0.325287, -1.181850, -2.686198, -0.844341, 1.570796, 1.896083],accel_mss,speed_ms,0,blend_radius_m)
    |   movel([0.324302, -1.182566, -2.685871, -0.843952, 1.570796, 1.895099],accel_mss,speed_ms,0,blend_radius_m)
    |   movel([0.323465, -1.182020, -2.686120, -0.844249, 1.570796, 1.894261],accel_mss,speed_ms,0,blend_radius_m)
    |   movel([0.322422, -1.181476, -2.686368, -0.844545, 1.570796, 1.893218],accel_mss,speed_ms,0,blend_radius_m)
    |   movel([0.321330, -1.181177, -2.686505, -0.844708, 1.570796, 1.892126],accel_mss,speed_ms,0,blend_radius_m)
    |   movel([0.320125, -1.181111, -2.686534, -0.844743, 1.570796, 1.890921],accel_mss,speed_ms,0,blend_radius_m)
    |   movel([0.318743, -1.181273, -2.686461, -0.844655, 1.570796, 1.889539],accel_mss,speed_ms,0,blend_radius_m)
    |   movel([0.317778, -1.181473, -2.686370, -0.844546, 1.570796, 1.888574],accel_mss,speed_ms,0,blend_radius_m)
    |   movel([0.316559, -1.181932, -2.686160, -0.844297, 1.570796, 1.887355],accel_mss,speed_ms,0,blend_radius_m)
    |   movel([0.315884, -1.182337, -2.685976, -0.844077, 1.570796, 1.886681],accel_mss,speed_ms,0,blend_radius_m)
    |   movel([0.314583, -1.183372, -2.685502, -0.843515, 1.570796, 1.885380],accel_mss,speed_ms,0,blend_radius_m)
    |   movel([0.313518, -1.184598, -2.684940, -0.842850, 1.570796, 1.884314],accel_mss,speed_ms,0,blend_radius_m)
    |   movel([0.313020, -1.185597, -2.684481, -0.842310, 1.570796, 1.883816],accel_mss,speed_ms,0,blend_radius_m)
    |   movel([0.313023, -1.185910, -2.684337, -0.842142, 1.570796, 1.883819],accel_mss,speed_ms,0,blend_radius_m)
    |   movel([0.313225, -1.186073, -2.684262, -0.842054, 1.570796, 1.884022],accel_mss,speed_ms,0,blend_radius_m)
    |   movel([0.313519, -1.186017, -2.684288, -0.842084, 1.570796, 1.884316],accel_mss,speed_ms,0,blend_radius_m)
    |   movel([0.313889, -1.185759, -2.684407, -0.842223, 1.570796, 1.884685],accel_mss,speed_ms,0,blend_radius_m)
    |   movel([0.314227, -1.185384, -2.684579, -0.842425, 1.570796, 1.885023],accel_mss,speed_ms,0,blend_radius_m)
    |   movel([0.314428, -1.184999, -2.684756, -0.842633, 1.570796, 1.885224],accel_mss,speed_ms,0,blend_radius_m)
    |   movel([0.314724, -1.184554, -2.684961, -0.842874, 1.570796, 1.885520],accel_mss,speed_ms,0,blend_radius_m)
    |   movel([0.315577, -1.183834, -2.685291, -0.843264, 1.570796, 1.886373],accel_mss,speed_ms,0,blend_radius_m)
    |   movel([0.316521, -1.183156, -2.685601, -0.843632, 1.570796, 1.887317],accel_mss,speed_ms,0,blend_radius_m)
    |   movel([0.317247, -1.182786, -2.685771, -0.843833, 1.570796, 1.888043],accel_mss,speed_ms,0,blend_radius_m)
    |   movel([0.318828, -1.182430, -2.685933, -0.844026, 1.570796, 1.889624],accel_mss,speed_ms,0,blend_radius_m)
    |   movel([0.320459, -1.182511, -2.685896, -0.843982, 1.570796, 1.891256],accel_mss,speed_ms,0,blend_radius_m)
    |   movel([0.321949, -1.182993, -2.685676, -0.843720, 1.570796, 1.892745],accel_mss,speed_ms,0,blend_radius_m)
    |   movel([0.323647, -1.184304, -2.685075, -0.843009, 1.570796, 1.894444],accel_mss,speed_ms,0,blend_radius_m)
    |   movel([0.324065, -1.184366, -2.685047, -0.842976, 1.570796, 1.894861],accel_mss,speed_ms,0,blend_radius_m)
    |   movel([0.324491, -1.184104, -2.685167, -0.843118, 1.570796, 1.895287],accel_mss,speed_ms,0,blend_radius_m)
    |   movel([0.325034, -1.183433, -2.685475, -0.843481, 1.570796, 1.895830],accel_mss,speed_ms,0,blend_radius_m)
    |   movel([0.325654, -1.182744, -2.685790, -0.843856, 1.570796, 1.896450],accel_mss,speed_ms,0,blend_radius_m)
    |   movel([0.326005, -1.182575, -2.685867, -0.843947, 1.570796, 1.896801],accel_mss,speed_ms,0,blend_radius_m)
    |   movel([0.327349, -1.182292, -2.685996, -0.844101, 1.570796, 1.898145],accel_mss,speed_ms,0,blend_radius_m)
    |   movel([0.328009, -1.182344, -2.685972, -0.844072, 1.570796, 1.898806],accel_mss,speed_ms,0,blend_radius_m)
    |   movel([0.329157, -1.182899, -2.685719, -0.843771, 1.570796, 1.899953],accel_mss,speed_ms,0,blend_radius_m)
    |   movel([0.330016, -1.184055, -2.685190, -0.843144, 1.570796, 1.900813],accel_mss,speed_ms,0,blend_radius_m)
    |   movel([0.330553, -1.185780, -2.684397, -0.842212, 1.570796, 1.901349],accel_mss,speed_ms,0,blend_radius_m)
    |   movel([0.330759, -1.187424, -2.683639, -0.841326, 1.570796, 1.901555],accel_mss,speed_ms,0,blend_radius_m)
    |   movel([0.330735, -1.188977, -2.682920, -0.840492, 1.570796, 1.901531],accel_mss,speed_ms,0,blend_radius_m)
    |   movel([0.330462, -1.190688, -2.682125, -0.839576, 1.570796, 1.901258],accel_mss,speed_ms,0,blend_radius_m)
    |   movel([0.329269, -1.195207, -2.680010, -0.837172, 1.570796, 1.900065],accel_mss,speed_ms,0,blend_radius_m)
    |   movel([0.329333, -1.195452, -2.679895, -0.837042, 1.570796, 1.900129],accel_mss,speed_ms,0,blend_radius_m)
    |   movel([0.329574, -1.195507, -2.679869, -0.837013, 1.570796, 1.900370],accel_mss,speed_ms,0,blend_radius_m)
    |   movel([0.329774, -1.195449, -2.679897, -0.837044, 1.570796, 1.900571],accel_mss,speed_ms,0,blend_radius_m)
    |   movel([0.330295, -1.195055, -2.680082, -0.837252, 1.570796, 1.901092],accel_mss,speed_ms,0,blend_radius_m)
    |   movel([0.330668, -1.194304, -2.680435, -0.837650, 1.570796, 1.901464],accel_mss,speed_ms,0,blend_radius_m)
    |   movel([0.331348, -1.191998, -2.681514, -0.838876, 1.570796, 1.902144],accel_mss,speed_ms,0,blend_radius_m)
    |   speed_ms = 0.005
    |   movel([0.331348, -1.145970, -2.656733, -0.909686, 1.570796, 1.902144],accel_mss,speed_ms,0,blend_radius_m)
    |   speed_ms = 1.000
    |   movel([0.331348, -1.145970, -2.656733, -0.909686, 1.570796, 1.902144],accel_mss,speed_ms,0,blend_radius_m)
    |   # Splitting Linear movement in 6 (instruction 8476: MoveL 8167)
    |   movel([0.331348, -1.112111, -2.635138, -0.965140, 1.570796, 1.902144],accel_mss,speed_ms,0,blend_radius_m)
    |   movel([0.331348, -1.082005, -2.612778, -1.017606, 1.570796, 1.902144],accel_mss,speed_ms,0,blend_radius_m)
    |   movel([0.331348, -1.055344, -2.589727, -1.067318, 1.570796, 1.902144],accel_mss,speed_ms,0,blend_radius_m)
    |   movel([0.331348, -1.031836, -2.566048, -1.114505, 1.570796, 1.902144],accel_mss,speed_ms,0,blend_radius_m)
    |   movel([0.331348, -1.011208, -2.541797, -1.159385, 1.570796, 1.902144],accel_mss,speed_ms,0,blend_radius_m)
    |   movel([0.331348, -0.993207, -2.517018, -1.202164, 1.570796, 1.902144],accel_mss,speed_ms,0,blend_radius_m)
    |   # End of main program
    | end
    | 
    | Machining1()
